(* IEC 61131-3 sources: Lasal/CPU_5344_V01/Class/inputsToSafety, 1 file *)

(* ---- inputsToSafety.st ---- *)
(*!
<Class
	Name               = "inputsToSafety"
	Revision           = "0.0"
	RealtimeTask       = "false"
	CyclicTask         = "true"
	DefCyclictime      = "10 ms"
	BackgroundTask     = "false"
	Sigmatek           = "false"
	OSInterface        = "false"
	HighPriority       = "false"
	Automatic          = "false"
	UpdateMode         = "Prescan"
	SharedCommandTable = "true"
	Objectsize         = "(360,720)">
	<Channels>
		<Server Name="ClassSvr" Visualized="false" Initialize="false" WriteProtected="true" Retentive="false"/>
		<Server Name="cmdInput1" Visualized="true" Initialize="false" WriteProtected="true" Retentive="false"/>
		<Server Name="cmdInput10" Visualized="true" Initialize="false" WriteProtected="true" Retentive="false"/>
		<Server Name="cmdInput2" Visualized="true" Initialize="false" WriteProtected="true" Retentive="false"/>
		<Server Name="cmdInput3" Visualized="true" Initialize="false" WriteProtected="true" Retentive="false"/>
		<Server Name="cmdInput4" Visualized="true" Initialize="false" WriteProtected="true" Retentive="false"/>
		<Server Name="cmdInput5" Visualized="true" Initialize="false" WriteProtected="true" Retentive="false"/>
		<Server Name="cmdInput6" Visualized="true" Initialize="false" WriteProtected="true" Retentive="false"/>
		<Server Name="cmdInput7" Visualized="true" Initialize="false" WriteProtected="true" Retentive="false"/>
		<Server Name="cmdInput8" Visualized="true" Initialize="false" WriteProtected="true" Retentive="false"/>
		<Server Name="cmdInput9" Visualized="true" Initialize="false" WriteProtected="true" Retentive="false"/>
		<Client Name="input1" Required="false" Internal="false"/>
		<Client Name="input10" Required="false" Internal="false"/>
		<Client Name="input2" Required="false" Internal="false"/>
		<Client Name="input3" Required="false" Internal="false"/>
		<Client Name="input4" Required="false" Internal="false"/>
		<Client Name="input5" Required="false" Internal="false"/>
		<Client Name="input6" Required="false" Internal="false"/>
		<Client Name="input7" Required="false" Internal="false"/>
		<Client Name="input8" Required="false" Internal="false"/>
		<Client Name="input9" Required="false" Internal="false"/>
	</Channels>
</Class>
*)
inputsToSafety : CLASS
  //Servers:
	ClassSvr 	: SvrChCmd_DINT;
	cmdInput1 	: SvrCh_DINT;
	cmdInput2 	: SvrCh_DINT;
	cmdInput3 	: SvrCh_DINT;
	cmdInput4 	: SvrCh_DINT;
	cmdInput5 	: SvrCh_DINT;
	cmdInput6 	: SvrCh_DINT;
	cmdInput7 	: SvrCh_DINT;
	cmdInput8 	: SvrCh_DINT;
	cmdInput9 	: SvrCh_DINT;
	cmdInput10 	: SvrCh_DINT;
  //Clients:
	input1 	: CltCh_DINT;
	input2 	: CltCh_DINT;
	input3 	: CltCh_DINT;
	input4 	: CltCh_DINT;
	input5 	: CltCh_DINT;
	input6 	: CltCh_DINT;
	input7 	: CltCh_DINT;
	input8 	: CltCh_DINT;
	input9 	: CltCh_DINT;
	input10 	: CltCh_DINT;
  //Variables:
  //Functions:

	FUNCTION VIRTUAL GLOBAL CyWork
		VAR_INPUT
			EAX 	: UDINT;
		END_VAR
		VAR_OUTPUT
			state (EAX) 	: UDINT := READY;
		END_VAR;
  //Tables:
	FUNCTION @STD
		VAR_OUTPUT
			ret_code	: CONFSTATES;
		END_VAR;
	FUNCTION GLOBAL TAB @CT_;
END_CLASS;

FUNCTION VIRTUAL GLOBAL inputsToSafety::CyWork
	VAR_INPUT
		EAX 	: UDINT;
	END_VAR
	VAR_OUTPUT
		state (EAX) 	: UDINT;(* := READY *)
	END_VAR

  input1 := input1.Read();
  input2 := input2.Read();
  input3 := input3.Read();
  input4 := input4.Read();
  input5 := input5.Read();
  input6 := input6.Read();
  input7 := input7.Read();
  input8 := input8.Read();
  input9 := input9.Read();
  input10 := input10.Read();

  cmdInput1:= input1;
  cmdInput2:= input2;
  cmdInput3:= input3;
  cmdInput4:= input4;
  cmdInput5:= input5;
  cmdInput6:= input6;
  cmdInput7:= input7;
  cmdInput8:= input8;
  cmdInput9:= input9;
  cmdInput10:= input10;

END_FUNCTION
